Staubli VAL3: lists.dtx

mdesc mNomSpeed
public string sString
